Universal Robots PolyScope program: ventosa_loop.urp

Program ventosa_loop (installation=ventosa directory=/programs/usbdisk createdIn=5.12.1.1101497 lastSavedIn=5.12.1.1101497 robotSerialNumber=20225300640)
Calibrated DH parameters: a=[-0.000125, -0.240482, -0.204397, 0.000169, -0.000135, 0]; d=[0.152056, 4.760815, 12.138494, -16.768367, 0.085457, 0.092357]; alpha=[1.570863, 0.008548, 0.003635, 1.571424, -1.571918, 0]; deltaTheta=[0, 0.167622, 0.124346, -0.291972, 0.000034, 0]
BeforeStart
  SafeHome (positionOptionType=SPEED_AND_ACCELERATION speed=1.047198 acceleration=1.396263 nextMotionTime=2)
  i := 0
  cnt_obj := 0
  dist_1 := 0.09
  dist_2 := 0.14
Robot Program (runOnlyOnce=false)
  Loop While (checkContinuously=false) expression=cnt_obj<2  and  i<3
    appro_1 := pose_trans(punt_ref_1, p[0-(dist_1*i),0,-0.04,0,0,0])
    MoveJ speed 60 deg/s, acceleration 80 deg/s^2 (useActiveTCP=true) feature=Base
      Waypoint Waypoint (Variable): variable=appro_1
    item_s1 := pose_trans(punt_ref_1, p[0-i*dist_1,0,0,0,0,0])
    MoveL speed 250 mm/s, acceleration 1200 mm/s^2 (useActiveTCP=true) feature=Base
      Waypoint Waypoint (Variable): variable=item_s1
    URCap Vacuum (Robotiq_Grippers, Robotiq Inc.) dataModel(Vacuum.Command.PumpAutoCloseDelayInMilliseconds=3000, Vacuum.Command.ShutOffDistance=5.0)
    MoveL speed 250 mm/s, acceleration 1200 mm/s^2 (useActiveTCP=true) feature=Base
      Waypoint Waypoint (Variable): variable=appro_1
    URCap Grip Check (Robotiq_Grippers, Robotiq Inc.) dataModel(ObjectDetectedKey=true, DimensionValidationKey=false, DimensionKey=100.0, DimensionDimensionPositiveGapKey=5.0, DimensionNegativeGapKey=5.0, GripperIdKey=1, ModelDefinedKey=true); state(isChildrenLocked=true)
      URCap If (Robotiq_Grippers, Robotiq Inc.)
        appro_s2 := pose_trans(punt_ref_2, p[0,0-cnt_obj*dist_2,0-0.04,0,0,0])
        MoveJ speed 60 deg/s, acceleration 80 deg/s^2 (useActiveTCP=true) feature=Base
          Waypoint Waypoint (Variable): variable=appro_s2
        item_s2 := pose_trans(punt_ref_2, p[0,-cnt_obj*dist_2,0,0,0,0])
        MoveL speed 250 mm/s, acceleration 1200 mm/s^2 (useActiveTCP=true) feature=Base
          Waypoint Waypoint (Variable): variable=item_s2
        URCap Vacuum (Robotiq_Grippers, Robotiq Inc.) dataModel(Vacuum.Command.Action=1, Vacuum.Command.PumpAutoCloseDelayInMilliseconds=3000, Vacuum.Command.ShutOffDistance=5.0)
        MoveL speed 250 mm/s, acceleration 1200 mm/s^2 (useActiveTCP=true) feature=Base
          Waypoint Waypoint (Variable): variable=appro_s2
        cnt_obj := cnt_obj+1
      URCap Else (Robotiq_Grippers, Robotiq Inc.)
        URCap Vacuum (Robotiq_Grippers, Robotiq Inc.) dataModel(Vacuum.Command.Action=1, Vacuum.Command.PumpAutoCloseDelayInMilliseconds=3000, Vacuum.Command.ShutOffDistance=5.0)
    i := i+1
  SafeHome (positionOptionType=SPEED_AND_ACCELERATION speed=1.047198 acceleration=1.396263 nextMotionTime=2)
  Halt
